FUNCTION_BLOCK FB_CO2Sensor EXTENDS FB_Sensor
VAR_INPUT
END_VAR
VAR_OUTPUT
	fCO2 : REAL; //measured CO2 concentration in ppm
END_VAR
VAR
	//I/O-Links
	CO2_IN AT %I* : INT;
	
END_VAR

METHOD GetState_AI : BOOL
VAR_INPUT
END_VAR
fCO2 :=  (CO2_IN / 32767.0)*2000; //conversion

//sensor state
sensorState.fValue := fCO2;
sensorState.sUnit := 'ppm';
END_METHOD

END_FUNCTION_BLOCK

(* stored: Version 1.1.0.1, ProductVersion 3.1.4024.6
   POU FB_CO2Sensor: Id {9b2af059-ccf9-478f-90e7-23670ad7fb61}, SpecialFunc None
   Method GetState_AI: Id {78bf2fd8-ac8b-4387-abaf-cc066038b9e9} *)
